// TIA Portal project "Set-Reset Uygulaması_2 (FBD)" (V18)

(* hardware
DEVICE "S7-1200 station_1"  S7-1200 Station
   slot 0: "Rack_0"  S7-1200 Rack  Rack  V1.0
   slot 1: "PLC_1"  CPU 1214C AC/DC/Rly  6ES7 214-1BG40-0XB0  V4.6
*)

// ===== PLC "PLC_1"  CPU 1214C AC/DC/Rly =====

VAR_GLOBAL   // PLC tag table "Default tag table"
   "Stop" AT %I0.0 : Bool;
   "Start_1" AT %I0.1 : Bool;
   "Start_2" AT %I0.2 : Bool;
   "Motor_1" AT %Q0.0 : Bool;
   "Start_3" AT %I0.3 : Bool;
   "Motor_2" AT %Q0.1 : Bool;
   "Motor_3" AT %Q0.2 : Bool;
   "Aşırı Akım Koruma" AT %I0.7 : Bool;
   "Motor_4" AT %Q0.3 : Bool;
   "Start_4" AT %I0.4 : Bool;
END_VAR

ORGANIZATION_BLOCK "Main"   // OB1, LAD, ProgramCycle
TITLE = "Main Program Sweep (Cycle)"
{ S7_Optimized_Access := 'TRUE' }
VERSION : 0.1
// Set-Reset Uygulamalarında 
// *Networkte önce set sonra reset varsa ve anahtarlara aynı anda basarsan RESET
// *Networkte önce reset sonra set varsa ve anahtarlara aynı anda basarsan SET
// DAİMA ALTTA OLAN ÇALIŞIR.
   VAR_INPUT
      Initial_Call : Bool;   // Initial call of this OB
      Remanence : Bool;   // =True, if remanent data are available
   END_VAR
BEGIN

REGION Network 1
   // Bu network için butonlara aynı anda basarsan alttaki satır yanı SET çalışacak.
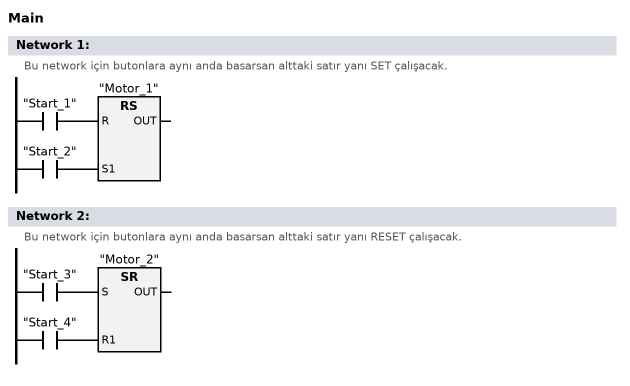
   RUNG wire#powerrail
      Contact( "Start_1" )
      S_RS(operand := "Motor_1", s1 := wire#w1)
   END_RUNG
   RUNG wire#powerrail
      Contact( "Start_2" )
   END_RUNG wire#w1
   // the same network as SCL:
   IF "Start_1" THEN
       "Motor_1" := FALSE;   // RS flip-flop
   END_IF;
   IF "Start_2" THEN "Motor_1" := TRUE; END_IF;
END_REGION

REGION Network 2
   // Bu network için butonlara aynı anda basarsan alttaki satır yanı RESET çalışacak.
   RUNG wire#powerrail
      Contact( "Start_3" )
      S_SR(operand := "Motor_2", r1 := wire#w1)
   END_RUNG
   RUNG wire#powerrail
      Contact( "Start_4" )
   END_RUNG wire#w1
   // the same network as SCL:
   IF "Start_3" THEN
       "Motor_2" := TRUE;   // SR flip-flop
   END_IF;
   IF "Start_4" THEN "Motor_2" := FALSE; END_IF;
END_REGION
END_ORGANIZATION_BLOCK